{attribute 'GeneratedUsingTerminal: KL3356'}
{attribute addProperty BoxType "KL3356"}
{attribute addProperty Id "Channel_1AT %Q*Channel_4E9D1E2D0"}
{attribute addProperty CRC "3758413026"}
{attribute addProperty Size "0"}
TYPE KL3356_E004D4E2 :
STRUCT
	{attribute addProperty Name "Channel_1"}
	Channel_1 : Channel_4E9D1E2D;
END_STRUCT
END_TYPE

(* stored: Version 1.2.0.0, ProductVersion 3.1.4024.9
   DUT KL3356_E004D4E2: Id {c0b67e17-1cd4-4b5c-896f-8792e93a32e4} *)
